(* PLC project SansNom, Inconnu SansNom 1 *)
(* stored: creationDateTime 2024-10-07T08:33:25, modificationDateTime 2024-10-07T08:33:25 *)

CONFIGURATION Config0
  RESOURCE Res0 ON PLC
  END_RESOURCE
END_CONFIGURATION
